ABB RobotStudio station: ProjectLab1.rsstnx

Station ProjectLab1 (saved by RobotStudio 24.1.10693.0)
Layout (positions relative to the parent item):
